TEXTLIST tlBottleTypes
  1 = 'A'
  2 = 'B'
  3 = 'C'
  0 = 'None'
   = ''
END_TEXTLIST

(* stored: Version 1.1.0.1, ProductVersion 3.1.4024.15
   TextList tlBottleTypes: Id {bf65fd5b-b35b-498a-b581-3fe8d6d238b2} *)
